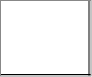
VISUALIZATION VISU_SystemButton_backup  // 92x77
VAR_IN_OUT
    widget : SystemButtonWidget;
END_VAR
    Rectangle (0,0 90x75), invisible if: widget.isNotOrange
    Rectangle (0,0 90x75), invisible if: widget.isNotGray
    Rectangle (0,0 90x75), invisible if: widget.isNotBlue
    Rectangle (0,0 90x75), invisible if: widget.isNotRed
    Rectangle (0,0 90x75), invisible if: widget.isNotGreen
    Rectangle (0,50 90x25), "%s", text variable: widget.name
    Image (25,10 40x40), image: VISU_SystemButtonImages.Home
        p84334746: widget.name
    Rectangle (0,0 90x75), invisible if: widget.notActivated
    Line (0,74) (90,74)
    Line (89,75) (89,0)
    Line (0,74) (0,0)
    Line (88,0) (0,0)
END_VISUALIZATION

(* stored: Version 1.1.0.1, ProductVersion 3.1.4019.2
   Visu VISU_SystemButton_backup: Id {a1ba98b2-fe5e-414b-ab18-732b39209d13} *)
